TYPE ST_SlideNest_CMD :
STRUCT
	
	MoveRight					: BOOL;				
	MoveLeft					: BOOL;		
	
END_STRUCT
END_TYPE

(* stored: Version 1.1.0.1, ProductVersion 3.1.4026.18
   DUT ST_SlideNest_CMD: Id {4d5ed30b-e653-45fe-b67e-82228baaa550} *)
